// TIA Portal V19 export
DATA_BLOCK "GET_Request_DB"   // DB10
// stored: InstanceOfName GET_Request, InstanceOfType FB
"GET_Request"
   // VAR_INPUT
   //    start : Bool;
   //    url : String;
   //    queryParams : String;
   // END_VAR
   // VAR_OUTPUT
   //    connected : Bool;
   //    done : Bool;
   //    busy : Bool;
   //    error : Bool;
   //    status : Word;
   //    diagnostics : "typeDiagnostics";
   //    responseCode : UInt;
   //    length : UDInt;
   // END_VAR
   // VAR_IN_OUT
   //    responseData : Array[*] of Char;
   // END_VAR
   // VAR
   //    hwID : HW_ANY;
   //    connID : CONN_OUC := 16#0003;
   //    keepConnection : Bool;
   //    userFields : Array[0..255] of Char;
   //    tls : "LHTTP_typeTLS";
   // END_VAR
BEGIN
END_DATA_BLOCK
